# B&R Automation Studio project CControl (part 2)

### Global.var
```iecst
VAR
	Boxen : {REDUND_UNREPLICABLE} fbBoxenKonfig; (*Baustein Trocknungsboxen*)
	Aktoren : {REDUND_UNREPLICABLE} typAktoren; (*Funktionsbausteine aller Aktoren (Ventilatoren, Trocknungsgeräte, Klappen, ...)*)
	Tarifabschaltung : {REDUND_UNREPLICABLE} fbTrockTarifabsch; (*Funktionsbaustein Tarifabschaltung*)
	Strombegrenzung : {REDUND_UNREPLICABLE} fbTrockStrombegr; (*Funktionsbaustein Strombegrenzung*)
END_VAR
VAR RETAIN
	Betriebsparameter : {REDUND_UNREPLICABLE} parAnlage; (*Betriebsparametersatz*)
END_VAR
VAR
	CONST_ZEIT_TESTPHASE : {REDUND_UNREPLICABLE} USINT := 3; (*max. Betriebsstunden, in denen der Kompressor am Luftentfeuchter gestartet werden kann, ohne dass die Mindestlaufzeit der Ölsumpfheizung abgelaufen ist (Für Inbetriebnahme Kältetechniker)*)
	gModul2Vorhanden : {REDUND_UNREPLICABLE} BOOL; (*Variable wird gesetzt, wenn eine Luftentfeuchter-Type mit 2 Kompressormodulen ausgewählt wird*)
	gAktModus : {REDUND_UNREPLICABLE} enumBetriebsmodus; (*Aktueller Schrittkettenzustand*)
	gStatusAnlage : {REDUND_UNREPLICABLE} statAnlage; (*Anlagenstatus*)
	gCmdAnlage : {REDUND_UNREPLICABLE} cmdAnlage; (*Anlagenkommandos*)
END_VAR
VAR RETAIN
	Nutzungsdaten : {REDUND_UNREPLICABLE} typNutzungsdaten; (*Struktur Betriebsstunden, Brennstoffleistung, etc...*)
END_VAR
VAR
	Echtzeit : {REDUND_UNREPLICABLE} typEchtzeit; (*Echtzeituhr*)
	Systeminfo : {REDUND_UNREPLICABLE} typSysteminfo; (*Struktur Systeminformationen (Batteriestatus, Hardwaremodule, etc...)*)
	DateTime : {REDUND_UNREPLICABLE} DATE_AND_TIME; (*Aktuelle Systemzeit*)
	VERSION : {REDUND_UNREPLICABLE} STRING[16] := 'V2.1.3'; (*Softwareversion*)
END_VAR
VAR RETAIN
	gMindestlaufzOelsumpfOk : {REDUND_UNREPLICABLE} BOOL; (*Variable wird gesetzt, wenn Mindestlaufzeit der Ölsumpfheiung abgelaufen ist.*)
END_VAR
VAR
	gAktuellesPasswort : {REDUND_UNREPLICABLE} UDINT; (*Aktuelles Passwort in der Visu (Benutzeranmeldung)*)
	gWerksparameterLaden : {REDUND_UNREPLICABLE} BOOL; (*Befehl Werksparametersatz laden*)
	gEnergiemessungModulOk : {REDUND_UNREPLICABLE} BOOL; (*Modulüberwachung Energiemessmodul (wird in den IO-Mappings zur Fehlergenerierung verwendet)*)
END_VAR
```

### versionsinfo.txt
```
##########################################################
LaTronic CControl 3.07, 4.07 & 4.07 Plus Versionshistorie
##########################################################

--------------------------------------------------------------------------------------------
Version 0.0.0	     	Initialversion			2022.05.19					RL
--------------------------------------------------------------------------------------------

--------------------------------------------------------------------------------------------
Version 0.0.1	     	new/change/fix			2022.06.01					RL
--------------------------------------------------------------------------------------------

Neu:
****
- Optionen für Verhalten der Ventilatoren bei Klappenumschaltungen hinzugefügt (Beide oder nur zuständigen Ventilator
bei Umschaltungen Boxenklappen, Umluftklappen und Bypassklappe).
- Option "Abluftklappe im Frischluftbetrieb immer offen" hinzugefügt (Abluftklappe öffnet im Frischluftbetrieb unabhängig von der
eingestellten Abluftfeuchte, wenn Klappe auf Automatik gestellt).
- Option "Alle Boxenklappen im Stillstand schließen" hinzugefügt.
- Trockengut "Mais" und "Getreide" hinzugefügt.
- VNC-Viewer bei allen Konfigurationen hinzugefügt.
- "Notbetrieb" für alle Boxen und Ventilatoren hinzugefügt (für Auskühlphase Warmluftofen). Boxenklappen und Ventilatoren bleiben aktiv,
bis Auskühlphase abgeschlossen ist.
- Funktion zum Kopieren der XML-Parametersätze auf einen USB-Stick hinzugefügt.
- Zusatztexte hinzugefügt, wenn Trocknungsgeräte wegen Tarifabschaltung aus sind (Vorlaufzeit Tarifabschaltung).
- Zoom für Trendkurven hinzugefügt.
- Hopfen und Kräuter bei Trockengütern hinzugefügt.
- Automatisches Laden der Werksparameter bei neuen Displays hinzugefügt.
- Französische Sprache hinzugefügt.
- Energiemessmodul in allen Hardwarekonfigurationen hinzugefügt.
- Trockengut "Holz" hinzugefügt (Visualisierung/Visu, hmiMain).
- Modulüberwachungen für alle Hardwarekonfigurationen hinzugefügt (IO/io307, io407, io407Plus).

Änderungen:
***********
- Wenn Strombegrenzung der Ventilatoren aktiv ist (Zeitfenster oder digitaler Eingang), geht der Luftentfeuchter bei Überschreiten
des max. Hochdrucks in den Standby-Betrieb (wie bei Klappenumschaltungen).
- Warnung "Entfeuchter Hochdruck max." wird nur generiert, wenn keine Strombegrenzung oder Klappenumschaltung aktiv ist.
- Nur Option "Abluftklappe" ODER "Abluftventilator" erlauben, beide Optionen sind nicht möglich.
- Beim Abschalten der Ventilatoren die Freigabe erst wegschalten, wenn Min-Drehzahl erreicht wurde.
- Buttons und Slider für Ausstattung und Konfiguration Aktoren Boxen sperren, wenn Benutzerebene < LASCO.
- Beim Wechsel von Betrieb auf AUS einer Box -> Arrays Zeitfenster Intervallbetrieb und Nachtrockung auf 0 setzen.
- Entfeuchter, Warmluftofen und Heizregister erst freigeben, wenn zuständiger Ventilator in Betrieb ist.
- Boxen können auch gestartet werden, wenn Summenfehler aktiv (Sperren Visu entfernt, Wechsel in Betriebsart "BETRIEB" trotz Summenfehler).
- Signal "cmdAnlage.FehlerStopp" entfernt (Trocknung kann trotz Fehler gestartet werden bzw. wird nicht mehr automatisch gestoppt).
- Ansteuerung Bypassklappe geändert (actionBetrieb).
- Skalierung Drehzahlvorgabe Kompressor Modul 1 und 2: Min auf "0" gesetzt. (IO/io307, io407Plus).
- Drehzahlvorgaben von FU Kompressor angepasst (Libaries/LascoEntfV2/fbEntfKompressor).
- Doppelmodul nur bei bei den Typen 7, 8, 9 und 10 (10 ist Reserve) (IO/aktorenMapping).
- Fehlermeldungen Entfeuchter Temperatur Eintritt Min/Max nur ausgeben, wenn Entfeuchter angefordert. (Alarmsystem/Alarm).
- Drehzahlvorgabe Heizregister auf Min. setzen, wenn Heizregister nicht freigegeben (Regelung/Leistung).
- Ventilatoren: Wenn eingestellte Drehzahl bei Klappenumschaltungen auf MIN (30%) -> Ventilator ausschalten (Libaries/LascoBoxen/fbBoxenVentKlappen).
- Automatikbetrieb von Abluftklappe auch im Stillstand aktivieren (Ablaufsteuerung/actionStillstand).
- Parameter "Hochdruck Max." und "Verzögerung Standy, wenn Hochdruck Max." bereits ab Benutzerebene "LASCO" einstellbar (Visualisierung/Visu).

Fehlerbehebungen:
*****************
- Indexe für Fehler, Systemmeldungen und Warnungen angepasst (für Filter bei historischen Alarmen).
- Fehler Laufzeitüberwachungen Boxenklappen nur generieren, wenn Klappe verwendet wird.
- Min/Max Werte bei Eingabefeldern Detailansicht Klappen hinzugefügt.
- Struktur "hmiAktuell" remanent deklariert, da ansonsten die Betriebsart der Box nach Stromausfall geändert wird.
- Taste "Datenaufzeichnung auf USB kopieren" zurücksetzen, wenn Kopiervorgang fertig.
- Diverse CSV-Variablen in Datencontainer aktualisiert.
- 4.07Plus: Signalart Luftgeschwindigkeitssensor auf 0-10V geändert.
- Restlaufzeit Ölsumpfheizung in hmiParameter speichern (war Betriebsparameter).
- 4.07 Plus: DO Freigabe Ventilator 2 von Ausgang 2 auf 1 geändert.
- Doppelbelegung von Funktionsbausteinen entfernt (Alarmsystem/Alarm).
- Zusatztext "Auskühlzeit Scheitholzofen" Fehlerbehebung (Visualisierung/hmiConnect).
- Zusatztext "Warten bis Entfeuchter im Stillstand" auch anzeigen, wenn Boxen pausiert werden (Visualisierung/hmiConnect).
- Status Umluftklappen "Aktiv" nur generieren, wenn Klappe in Ausstattung vorhanden (IO/aktorenMapping).
- Digitale Eingänge "diOeldruckKompressorModul2" und "diKopftemperaturKompressorModul2" ausgetauscht (IO/io407Plus).
- Eingang "BetriebsmeldungVent" von Kompressor Modul 2 korrigiert (IO/aktorenMapping).
- "StoerungOut" von Funktionsbaustein "fbEntfKompressor" nicht automatisch rücksetzen, muss manuell quittiert werden (Libaries/LaEntfV2/fbEntfKompressor).
- Digialen Eingang "BetriebsmldgKompressorMod1" im IO-Test korrigiert (IO/io407Plus).
- 3.07: Je nach Ausstattung Analogeingänge und Statuseingänge als Dachluft- oder Frischluftsensor skalieren (IO/io307).

--------------------------------------------------------------------------------------------
Version 1.0.0	     	Erstversion Auslieferung		2022.06.22					RL
--------------------------------------------------------------------------------------------

--------------------------------------------------------------------------------------------
Version 1.1.0	     	new/fix/change					2022.09.22					RL
--------------------------------------------------------------------------------------------

Neu:
****
- Slowenische Sprache hinzugefügt (Visualisierung).
- Laden und Erstellen eines Parametersatzes sperren, wenn Filename "307Werk", "407Werk" oder "407PlusWerk" ist (Visualisierung/Visu).

Änderungen:
***********
- Die letzten 100 Ereignisse in der Alarmhistorie werden remanent aufgezeichnet (Visualisierung/Visu).

Fehlerbehebungen:
*****************
- Temperatur Austritt Entfeuchter: Falsch angehängten Wert in Visu korrigiert (Visualisierung/hmiMain).

TODO:
*****
- Verzögerungszeit Umschaltung Klappen, bis Endlage erreicht wurde?

--------------------------------------------------------------------------------------------
Version 1.1.1	     	fix								2022.09.22					RL
--------------------------------------------------------------------------------------------

Fehlerbehebungen:
*****************
- Bei Anlagen mit Bypassklappe: Freigabe Entfeuchter war von Betrieb des zuständigen Ventilators abhängig. Dadurch war die Freigabe des Kompressors immer nur solange
vorhanden, bis die Bypassklappe umgeschaltet wurde (ständiges hin- und herschalten der Klappen). Geändert, dass die Kompressor-Freigabe erhalten bleibt, wenn die Ventilatoren
kurzzeitig zum Umschalten der Klappen ausgeschaltet werden (Ablaufsteuerung/Ablaufstrg/actionBetrieb).

--------------------------------------------------------------------------------------------
Version 1.1.2	     	new								2023.05.03					RL
--------------------------------------------------------------------------------------------

Neu:
****
- Sensor Kanaldruck für Konfiguration 3.07 hinzugefügt (IO/io307).

--------------------------------------------------------------------------------------------
Version 1.2.0	     	new/change						2023.05.26					RL
--------------------------------------------------------------------------------------------

Neu:
****
- Neue Visualisierung für CControl 3.04 hinzugefügt (PPC30 4 Zoll).
- Hardwarekonfiguration & IO-mapping für CControl 3.04 hinzugefügt.
- Ausgänge öffnen/schliessen für Klappenansteuerungen (Umluftklappen, Bypassklappe, Abluftklappe, ...) hinzugefügt.
- Inselbetrieb für Luftentfeuchter hinzugefügt.

Änderungen:
***********
- Statuseingang "rel. Feuchte MAX" bei allen Feuchte/Temperaturfühlern für Fehlergenerierung entfernt (führt ansonsten zu Fehler, wenn rel. Feuchte tatsächlich bei 100% ist) (Alarmsystem/Alarm)

--------------------------------------------------------------------------------------------
Version 2.0.0	     	new/change						2024.07.04					RL
--------------------------------------------------------------------------------------------

Neu:
****
- Konfiguration für HB4000 & HB3000 hinzugefügt.
- Betriebsmodus "Dauerbetrieb" in "Automatik" umbenannt. Bei Anlagen ohne Luftaufbereitung (Kaltbelüftungen) wechselt die Box
bei schlechter Witterung in einen Puls/Pausebetrieb (wie bei HB3000/HB4000). Die Bestimmung der Witterungsverhältnisse kann für jede
Box seperat eingestellt werden.
- Entfeuchter Fremdgerät hinzugefügt (Ansteuerung von Frigopol/Baier Luftentfeuchtern).
- Option für Stellung Umluftklappen im Stillstand (Frischluft oder Umluft), wenn Umluftklappen im Automatikbetrieb sind.
- Option "Endlagen" für alle Klappenantriebe (ausgenommen Abluftklappe) hinzugefügt. Wird die Option ausgeschaltet (keine Endlagen vorhanden), wird über die
eingestellte Laufzeit der Klappe die Fahrt simuliert (Ventilator bleibt für die Laufzeit ausgeschaltet/reduziert).

Änderungen:
***********
- Im Stillstand Umluftklappen & Abluftklappe nicht automatisch umschalten (Ablaufsteuerung, Ablaufstrg/actionBetrieb).
- Default-Gateway als DEV1-Port verwenden (war fix auf 10.0.0.1 eingestellt) (Sitemanager/Sitemanager).
- Parameter "Einschaltverzögerung Entfeuchter" von 30 auf 120 Sekunden im Standardparametersatz aller Entfeuchtersteuerungen geändert (lt. Werner).

TODO:
*****
- Übersetzungen ergänzen (Aktuell nur Deutsch und Englisch verfügbar)
- Visu 3.04
- Standardparameter restliche Steuerungen

--------------------------------------------------------------------------------------------
Version 2.1.0	     	new/change						2024.12.02					RL
--------------------------------------------------------------------------------------------

Neu:
****
- Option Stellung Umluftklappen im Stillstand: Stellung kann für Klappe 1 und 2 separat eingestellt werden.
- Konfiguration für CControl 2.07 hinzugefügt.

Änderungen:
***********
- Schlechtwetterbetrieb: Anstatt der Boxenlaufzeit (in Stunden) wird die aktuelle Stufe durch die Trockengutfeuchte (%) bestimmt (manuelle Eingabe durch Bediener).

--------------------------------------------------------------------------------------------
Version 2.1.1	     	new/change						2025.05.07					RIG
--------------------------------------------------------------------------------------------

Änderungen:
***********
- Bugfix - Bei der Karte X20CM8281f war die Modulueberwachung aktiviert. Dies fuehrte dazu das die Steuerung nicht hochgefahren ist und beim Booten im Servicemodus haengen blieb.

--------------------------------------------------------------------------------------------
Version 2.1.2	     	new/change						2025.05.15					RIG
--------------------------------------------------------------------------------------------

Änderungen:
***********
- Bugfix - Fehler Betriebsmeldung "Entfeuchter Fremdgerät" wurde gesetzt obwohl Fremdgeraet nicht aktiviert war

--------------------------------------------------------------------------------------------
Version 2.1.3	     	new/change						2025.06.12					RIG
--------------------------------------------------------------------------------------------

Neu:
****
- Parametersaetze fuer 3.04 und 3.07 erstellt. Wurden aus 4.07 kopiert!
- Registerflache <Property ID="[2]" DataType="REAL" Value="3.3" /> von 3.8 auf 3.3 geaendert. Laut Werner war das schon immer falsch.

Änderungen:
***********
- Bugfix - Klappenansteuerung Anzugsverzoegerung fuer oeffnen und schliessen der Klappen eingebaut. Dient dazu das andere Relaise abfallen zu lassen bevor das andere geschaltet wird. Verhindert Doppelansteuerung.
```

### Program Logical/Alarmsystem/Alarm

#### AlarmCyclic.st
```iecst
PROGRAM _INIT

	init	:= FALSE;

END_PROGRAM

PROGRAM _CYCLIC

	//Sekundentick generieren
	//=======================
	eUhr(Freigabe:= TRUE);
	fbLascoZdxx_0(IN := eUhr.Sekunde);
	sekTick	:= fbLascoZdxx_0.Q;

	//Fehlergenerierung eingeschaltet *****************************************************************************************************************************************************************
	IF init THEN

		//=======================================================================================================================================================
		//FEHLER ------------------------------ FEHLER ------------------------------ FEHLER ------------------------------ FEHLER ------------------------------
		//=======================================================================================================================================================

		//00) Fehler Absicherung 24VDC
		alarmFehler[FEHLER_24VDC]			:= NOT di24VDCinternIstOk;

		//01) Fehler FU Kompressor Modul 1
		alarmFehler[FEHLER_FU_KOMPRESSOR_MODUL1]	:= Aktoren.KompressorModul1.StoerungOut;

		//02) Fehler FU Kompressor Modul 2
		alarmFehler[FEHLER_FU_KOMPRESSOR_MODUL2]	:= Aktoren.KompressorModul2.StoerungOut;

		//03) Fehler Betriebsmeldung Kompressor Modul 1
		fbLascoFehl_0(FehlerIn := doKompressorEinModul1 AND NOT diBetriebsmldgKompressorModul1,
		VerzZeit := Betriebsparameter.Allgemein.VerzoegerungFehler, Quit := hmiButtons.QuitFehler, Tick := sekTick, Mode := 1);
		alarmFehler[FEHLER_BETRIEBSMLDG_KOMPR_MOD1]	:= fbLascoFehl_0.FehlerOut;

		//04) Fehler Betriebsmeldung Kompressor Modul 2
		fbLascoFehl_1(FehlerIn := gModul2Vorhanden AND doKompressorEinModul2 AND NOT diBetriebsmldgKompressorModul2,
		VerzZeit := Betriebsparameter.Allgemein.VerzoegerungFehler, Quit := hmiButtons.QuitFehler, Tick := sekTick, Mode := 1);
		alarmFehler[FEHLER_BETRIEBSMLDG_KOMPR_MOD2]	:= fbLascoFehl_1.FehlerOut;

		//05) Fehler Betriebsmeldung Ventilator 1
		fbLascoFehl_2(FehlerIn := Aktoren.VentUndKlappen.FehlerFuVentilator1,
		VerzZeit := 0, Quit := hmiButtons.QuitFehler, Tick := sekTick, Mode := 1);
		alarmFehler[FEHLER_BETRIEBSMLDG_VENTILATOR1]	:= fbLascoFehl_2.FehlerOut;

		//06) Fehler Betriebsmeldung Ventilator 2
		fbLascoFehl_3(FehlerIn := Aktoren.VentUndKlappen.FehlerFuVentilator2,
		VerzZeit := 0, Quit := hmiButtons.QuitFehler, Tick := sekTick, Mode := 1);
		alarmFehler[FEHLER_BETRIEBSMLDG_VENTILATOR2]	:= fbLascoFehl_3.FehlerOut;

		//07) Fehler Betriebsmeldung Abluftventilator
		fbLascoFehl_4(FehlerIn := Aktoren.Abluftventilator.FehlerOut,
		VerzZeit := 0, Quit := hmiButtons.QuitFehler, Tick := sekTick, Mode := 1);
		alarmFehler[FEHLER_BETRIEBSMLDG_ABLUFTVENT]	:= fbLascoFehl_4.FehlerOut;

		//08) Fehler Hochdruck Modul 1
		fbLascoFehl_5(FehlerIn :=  Betriebsparameter.Ausstattung.Entfeuchter AND NOT diHochdruckOkModul1, VerzZeit := 0,
		Quit := hmiButtons.QuitFehler, Tick := sekTick, Mode := 0);
		alarmFehler[FEHLER_HOCHDRUCK_MODUL1]			:= fbLascoFehl_5.FehlerOut;

		//09) Fehler Hochdruck Modul 2
		fbLascoFehl_6(FehlerIn :=  Betriebsparameter.Ausstattung.Entfeuchter AND gModul2Vorhanden AND NOT diHochdruckOkModul2, VerzZeit := 0,
		Quit := hmiButtons.QuitFehler, Tick := sekTick, Mode := 0);
		alarmFehler[FEHLER_HOCHDRUCK_MODUL2]			:= fbLascoFehl_6.FehlerOut;

		//10) Fehler Niederdruck Modul 1
		fbLascoFehl_7(FehlerIn := Betriebsparameter.Ausstattung.Entfeuchter AND NOT diNiederdruckOkModul1, VerzZeit := 0,
		Quit := hmiButtons.QuitFehler, Tick := sekTick, Mode := 0);
		alarmFehler[FEHLER_NIEDERDRUCK_MODUL1]			:= fbLascoFehl_7.FehlerOut;

		//11) Fehler Niederdruck Modul 2
		fbLascoFehl_8(FehlerIn := Betriebsparameter.Ausstattung.Entfeuchter AND gModul2Vorhanden AND NOT diNiederdruckOkModul2,
		VerzZeit := 0, Quit := hmiButtons.QuitFehler, Tick := sekTick, Mode := 0);
		alarmFehler[FEHLER_NIEDERDRUCK_MODUL2]			:= fbLascoFehl_8.FehlerOut;

		//12) Fehler Öldruck Kompressor Modul 1
		fbLascoFehl_9(FehlerIn := Betriebsparameter.Ausstattung.Entfeuchter AND NOT diOeldruckKompressorModul1,
		VerzZeit := 0, Quit := hmiButtons.QuitFehler, Tick := sekTick, Mode := 0);
		alarmFehler[FEHLER_OELDRUCK_KOMPR_MOD1]			:= fbLascoFehl_9.FehlerOut;

		//13) Fehler Öldruck Kompressor Modul 2
		fbLascoFehl_10(FehlerIn := Betriebsparameter.Ausstattung.Entfeuchter AND gModul2Vorhanden AND NOT diOeldruckKompressorModul2,
		VerzZeit := 0, Quit := hmiButtons.QuitFehler, Tick := sekTick, Mode := 0);
		alarmFehler[FEHLER_OELDRUCK_KOMPR_MOD2]			:= fbLascoFehl_10.FehlerOut;

		//14) Fehler Kopftemperatur Kompressor Modul 1
		fbLascoFehl_11(FehlerIn := Betriebsparameter.Ausstattung.Entfeuchter AND NOT diKopftempKompressorModul1,
		VerzZeit := 0, Quit := hmiButtons.QuitFehler, Tick := sekTick, Mode := 0);
		alarmFehler[FEHLER_KOPFTEMP_KOMPR_MOD1]			:= fbLascoFehl_11.FehlerOut;

		//15) Fehler Kopftemperatur Kompressor Modul 2
		fbLascoFehl_12(FehlerIn := Betriebsparameter.Ausstattung.Entfeuchter AND gModul2Vorhanden AND NOT diKopftempKompressorModul2,
		VerzZeit := 0, Quit := hmiButtons.QuitFehler, Tick := sekTick, Mode := 0);
		alarmFehler[FEHLER_KOPFTEMP_KOMPR_MOD2]			:= fbLascoFehl_12.FehlerOut;

		//16) Fehler Vollschutz Kompressor Modul 1
		fbLascoFehl_13(FehlerIn := Betriebsparameter.Ausstattung.Entfeuchter AND NOT diVollschutzKompressorModul1,
		VerzZeit := 0, Quit := hmiButtons.QuitFehler, Tick := sekTick, Mode := 0);
		alarmFehler[FEHLER_VOLLSCHUTZ_KOMPR_MOD1]			:= fbLascoFehl_13.FehlerOut;

		//17) Fehler Vollschutz Kompressor Modul 2
		fbLascoFehl_14(FehlerIn := Betriebsparameter.Ausstattung.Entfeuchter AND gModul2Vorhanden AND NOT diVollschutzKompressorModul2,
		VerzZeit := 0, Quit := hmiButtons.QuitFehler, Tick := sekTick, Mode := 0);
		alarmFehler[FEHLER_VOLLSCHUTZ_KOMPR_MOD2]			:= fbLascoFehl_14.FehlerOut;

		//18) Fehler Betriebsmeldung Warmluftofen
		alarmFehler[FEHLER_BETRIEBSMLDG_WARMLUFTOFEN]	:= Aktoren.Warmluftofen.FehlerBetriebsmeldungOut;

		//19) Fehler Betriebsmeldung Notstromaggregat
		alarmFehler[FEHLER_BETRIEBSMLDG_NOTSTROM]		:= Aktoren.Notstromaggregat.FehlerOut;

		//20 - 31) Sensoren
		fbLascoFehl_15(FehlerIn := ((*diStatusFrischluftFeuchteMax OR *)diStatusFrischluftFeuchteMin OR diStatusFrischluftTempMax OR diStatusFrischluftTempMin) AND
		Betriebsparameter.Ausstattung.SensorFrischluft, VerzZeit := Betriebsparameter.Allgemein.VerzoegerungFehler,
		Quit := hmiButtons.QuitFehler, Tick := sekTick, Mode := 1);
		alarmFehler[FEHLER_SENSOR_FRISCHLUFT]	:= fbLascoFehl_15.FehlerOut;

		fbLascoFehl_16(FehlerIn := ((*diStatusDachluftFeuchteMax OR *)diStatusDachluftFeuchteMin OR diStatusDachluftTempMax OR diStatusDachluftTempMin) AND
		Betriebsparameter.Ausstattung.SensorDachluft, VerzZeit := Betriebsparameter.Allgemein.VerzoegerungFehler,
		Quit := hmiButtons.QuitFehler, Tick := sekTick, Mode := 1);
		alarmFehler[FEHLER_SENSOR_DACHLUFT]	:= fbLascoFehl_16.FehlerOut;

		fbLascoFehl_17(FehlerIn := ((*diStatusTrockenluftFeuchteMax OR *)diStatusTrockenluftFeuchteMin OR diStatusTrockenluftTempMax OR diStatusTrockenluftTempMin) AND
		Betriebsparameter.Ausstattung.SensorTrockenluft, VerzZeit := Betriebsparameter.Allgemein.VerzoegerungFehler,
		Quit := hmiButtons.QuitFehler, Tick := sekTick, Mode := 1);
		alarmFehler[FEHLER_SENSOR_TROCKENLUFT]	:= fbLascoFehl_17.FehlerOut;

		fbLascoFehl_18(FehlerIn := ((*diStatusAbluftFeuchteMax OR *)diStatusAbluftFeuchteMin OR diStatusAbluftTempMax OR diStatusAbluftTempMin) AND
		Betriebsparameter.Ausstattung.SensorAbluft,VerzZeit := Betriebsparameter.Allgemein.VerzoegerungFehler,
		Quit := hmiButtons.QuitFehler, Tick := sekTick, Mode := 1);
		alarmFehler[FEHLER_SENSOR_ABLUFT]	:= fbLascoFehl_18.FehlerOut;

		fbLascoFehl_19(FehlerIn := Betriebsparameter.Ausstattung.Entfeuchter AND
		((*diStatusEintrittFeuchteMax OR *)diStatusEintrittFeuchteMin OR diStatusEintrittTempMax OR diStatusEintrittTempMin),
		VerzZeit := Betriebsparameter.Allgemein.VerzoegerungFehler, Quit := hmiButtons.QuitFehler, Tick := sekTick, Mode := 1);
		alarmFehler[FEHLER_SENSOR_EINTRITT]	:= fbLascoFehl_19.FehlerOut;

		alarmFehler[FEHLER_SENSOR_AUSTRITT]	:= FALSE;	//Fehler Sensor Austritt nur als Warnung generieren

		fbLascoFehl_20(FehlerIn := (diStatusLuftgeschwDrahtbruch OR diStatusLuftgeschwMax OR diStatusLuftgeschwMin) AND Betriebsparameter.Ausstattung.SensorLuftgeschwindigkeit,
		VerzZeit := Betriebsparameter.Allgemein.VerzoegerungFehler, Quit := hmiButtons.QuitFehler, Tick := sekTick, Mode := 1);
		alarmFehler[FEHLER_SENSOR_LUFTGESCHW]	:= fbLascoFehl_20.FehlerOut;

		fbLascoFehl_21(FehlerIn := (diStatusDifferenzdruckMax OR diStatusDifferenzdruckMin) AND Betriebsparameter.Ausstattung.SensorKanaldruck,
		VerzZeit := Betriebsparameter.Allgemein.VerzoegerungFehler, Quit := hmiButtons.QuitFehler, Tick := sekTick, Mode := 1);
		alarmFehler[FEHLER_SENSOR_KANALDRUCK]	:= fbLascoFehl_21.FehlerOut;

		fbLascoFehl_22(FehlerIn := Betriebsparameter.Ausstattung.Entfeuchter AND (diStatusNiederdruckMaxMod1 OR diStatusNiederdruckMinMod1),
		VerzZeit := Betriebsparameter.Allgemein.VerzoegerungFehler, Quit := hmiButtons.QuitFehler, Tick := sekTick, Mode := 1);
		alarmFehler[FEHLER_SENSOR_NIEDERDRUCK_MOD1]	:= fbLascoFehl_22.FehlerOut;

		fbLascoFehl_23(FehlerIn := Betriebsparameter.Ausstattung.Entfeuchter AND gModul2Vorhanden AND (diStatusNiederdruckMaxMod2 OR diStatusNiederdruckMinMod2),
		VerzZeit := Betriebsparameter.Allgemein.VerzoegerungFehler, Quit := hmiButtons.QuitFehler, Tick := sekTick, Mode := 1);
		alarmFehler[FEHLER_SENSOR_NIEDERDRUCK_MOD2]	:= fbLascoFehl_23.FehlerOut;

		fbLascoFehl_24(FehlerIn := Betriebsparameter.Ausstattung.Entfeuchter AND (diStatusHochdruckMaxMod1 OR diStatusHochdruckMinMod1),
		VerzZeit := Betriebsparameter.Allgemein.VerzoegerungFehler, Quit := hmiButtons.QuitFehler, Tick := sekTick, Mode := 1);
		alarmFehler[FEHLER_SENSOR_HOCHDRUCK_MOD1]	:= fbLascoFehl_24.FehlerOut;

		fbLascoFehl_25(FehlerIn := Betriebsparameter.Ausstattung.Entfeuchter AND gModul2Vorhanden AND (diStatusHochdruckMaxMod2 OR diStatusHochdruckMinMod2),
		VerzZeit := Betriebsparameter.Allgemein.VerzoegerungFehler, Quit := hmiButtons.QuitFehler, Tick := sekTick, Mode := 1);
		alarmFehler[FEHLER_SENSOR_HOCHDRUCK_MOD2]	:= fbLascoFehl_25.FehlerOut;

		//32) Fehler Endlagen Bypassklappe
		alarmFehler[FEHLER_ENDLAGEN_BYPASSKLAPPE]		:= Aktoren.VentUndKlappen.FehlerLaufzeitBypass AND Betriebsparameter.Ausstattung.Bypassklappe;

		//33) Fehler Endlagen Umschaltklappe 1
		alarmFehler[FEHLER_ENDLAGEN_UMSCHALTKLAPPE1]	:= Aktoren.VentUndKlappen.FehlerLaufzeitUmschaltkl1 AND Betriebsparameter.Ausstattung.Umschaltklappe1;

		//34) Fehler Endlagen Umschaltklappe 2
		alarmFehler[FEHLER_ENDLAGEN_UMSCHALTKLAPPE2]	:= Aktoren.VentUndKlappen.FehlerLaufzeitUmschaltkl2 AND Betriebsparameter.Ausstattung.Umschaltklappe2;

		//35) Fehler Endlagen Boxenklappe 1
		alarmFehler[FEHLER_ENDLAGEN_BOXENKLAPPE_1]		:= Aktoren.VentUndKlappen.FehlerLaufzeitKlappeBox1;

		//36) Fehler Endlagen Boxenklappe 2
		alarmFehler[FEHLER_ENDLAGEN_BOXENKLAPPE_2]		:= Aktoren.VentUndKlappen.FehlerLaufzeitKlappeBox2;

		//37) Fehler Endlagen Boxenklappe 3
		alarmFehler[FEHLER_ENDLAGEN_BOXENKLAPPE_3]		:= Aktoren.VentUndKlappen.FehlerLaufzeitKlappeBox3;

		//38) Fehler Endlagen Boxenklappe 4
		alarmFehler[FEHLER_ENDLAGEN_BOXENKLAPPE_4]		:= Aktoren.VentUndKlappen.FehlerLaufzeitKlappeBox4;

		//39) Fehler Endlagen Boxenklappe 5
		alarmFehler[FEHLER_ENDLAGEN_BOXENKLAPPE_5]		:= Aktoren.VentUndKlappen.FehlerLaufzeitKlappeBox5;

		//40) Fehler Endlagen Boxenklappe 6
		alarmFehler[FEHLER_ENDLAGEN_BOXENKLAPPE_6]		:= Aktoren.VentUndKlappen.FehlerLaufzeitKlappeBox6;

		//41) Fehler Endlagen Abluftklappe
		alarmFehler[FEHLER_ENDLAGEN_ABLUFTKLAPPE]		:= Aktoren.Abluftklappe.FehlerLaufzeit;

		//42) Fehler Temperatur Eintritt zu hoch
		alarmFehler[FEHLER_EINTRITT_TEMP_ZU_HOCH]		:= (gStatusAnlage.EintrittTemperatur > Betriebsparameter.Kompressor1.EintrittTempMax) AND
		Betriebsparameter.Ausstattung.Entfeuchter AND Boxen.FreigabeLuftentfeuchter;

		//43) Fehler Temperatur Eintritt zu niedrig
		alarmFehler[FEHLER_EINTRITT_TEMP_ZU_NIEDRIG]	:= (gStatusAnlage.EintrittTemperatur < Betriebsparameter.Kompressor1.EintrittTempMin) AND
		Betriebsparameter.Ausstattung.Entfeuchter AND Boxen.FreigabeLuftentfeuchter;

		//44) Fehler Laufzeit Pumpdown Kompressor Modul 1
		alarmFehler[FEHLER_LZ_PUMPDOWN_MOD1]			:= Aktoren.KompressorModul1.FehlerPumpdown;

		//45) Fehler Laufzeit Pumpdown Kompressor Modul 2
		alarmFehler[FEHLER_LZ_PUMPDOWN_MOD2]			:= Aktoren.KompressorModul2.FehlerPumpdown AND gModul2Vorhanden;

		//46) Drehfeldüberwachung (Nur bei 3.04 Plus vorhanden)
		IF hmiStatus.NameSteuerung = 3 THEN
			alarmFehler[FEHLER_DREHFELD]	:= NOT diDrehfeldIstKorrekt AND NOT alarmSystem[FEHLER_KOMMUNIKATION_DISPLAY_IO];
		ELSE
			alarmFehler[FEHLER_DREHFELD]	:= FALSE;
		END_IF

		//47) Störmeldung Entfeuchter Fremdgeräte
		fbLascoFehl_29(FehlerIn := Betriebsparameter.Ausstattung.EntfeuchterFremd AND diEntfeuchterFremdStoerung,
		VerzZeit := Betriebsparameter.Allgemein.VerzoegerungFehler, Quit := hmiButtons.QuitFehler, Tick := sekTick, Mode := 2);
		alarmFehler[FEHLER_ENTF_FREMD_STOERMELDUNG]			:= fbLascoFehl_29.FehlerOut;

		//48) Fehler Betriebsmeldung Entfeuchter Fremdgerät
		alarmFehler[FEHLER_ENTF_FREMD_BETRMLDG]			:= Betriebsparameter.Ausstattung.EntfeuchterFremd AND Aktoren.EntfeuchterFremd.FehlerBetriebsmldg; //V2.1.2

		//=======================================================================================================================================================
		//WARNUNGEN ------------------------------ WARNUNGEN ------------------------------ WARNUNGEN ------------------------------ WARNUNGEN ------------------
		//=======================================================================================================================================================

		//00) Warnung wenn Hochdruck Modul 1 zu hoch (Register verschmutzt, Ansaugtemperatur zu hoch oder zu wenig Luftmenge
		fbLascoFehl_26(FehlerIn := gStatusAnlage.Betrieb AND (gStatusAnlage.HochdruckModul1 > Betriebsparameter.Kompressor1.HochdruckMax) AND NOT
		Aktoren.KompressorModul1.KlappenumschaltungAkiv,
		VerzZeit := Betriebsparameter.Allgemein.VerzoegerungWarnungen, Quit := hmiButtons.QuitFehler, Tick := sekTick, Mode := 0);
		alarmWarnung[WARNUNG_HOCHDRUCK_MAX_MOD1]	:= fbLascoFehl_26.FehlerOut;

		//01) Warnung wenn Hochdruck Modul 2 zu hoch (Register verschmutzt, Ansaugtemperatur zu hoch oder zu wenig Luftmenge
		fbLascoFehl_27(FehlerIn := gModul2Vorhanden AND gStatusAnlage.Betrieb AND
		(gStatusAnlage.HochdruckModul2 > Betriebsparameter.Kompressor1.HochdruckMax) AND NOT Aktoren.KompressorModul2.KlappenumschaltungAkiv,
		VerzZeit := Betriebsparameter.Allgemein.VerzoegerungWarnungen, Quit := hmiButtons.QuitFehler, Tick := sekTick, Mode := 0);
		alarmWarnung[WARNUNG_HOCHDRUCK_MAX_MOD2]	:= fbLascoFehl_27.FehlerOut;

		//02) Warnung Sensor Austritt
		fbLascoFehl_28(FehlerIn := diStatusAustrittFeuchteMax OR diStatusAustrittFeuchteMin OR diStatusAustrittTempMax OR diStatusAustrittTempMin,
		VerzZeit := Betriebsparameter.Allgemein.VerzoegerungFehler, Quit := hmiButtons.QuitFehler, Tick := sekTick, Mode := 1);
		alarmWarnung[WARNUNG_SENSOR_AUSTRITT]	:= fbLascoFehl_28.FehlerOut;

		//==================================================================================================================================================================
		//Fehlerausgang
		//==================================================================================================================================================================

		IF (gStatusAnlage.Betrieb OR gAktModus = STILLSTAND) THEN
			doTrocknungStoerung 	:= gStatusAnlage.Fehler.SummeFehler;
		ELSE
			doTrocknungStoerung	:= FALSE;
		END_IF

	END_IF

	//00 - 04 Systemfehler

	//alarmSystem[FEHLER_KOMMUNIKATION_DISPLAY_IO]	:= ; Wird in den IO-Mappings erzeugt.
	alarmSystem[FEHLER_IO_TEST_NICHT_FERTIG]		:= NOT Nutzungsdaten.Allgemein.IoTestAbgeschlossen;

	//Fehlerquittierung rücksetzen
	TON_Fehlerquittierung.IN	:= hmiButtons.QuitFehler;
	TON_Fehlerquittierung.PT	:= UDINT_TO_TIME(CONST_VERZ_QUIT);
	TON_Fehlerquittierung();

	IF (TON_Fehlerquittierung.Q) THEN
		hmiButtons.QuitFehler	:= FALSE;
	END_IF

	//Gruppenalarme bilden
	//********************

	gStatusAnlage.Fehler.SummeFehler := FALSE;
	gStatusAnlage.Fehler.FehlerNr	 := 0;
	ilen := (SIZEOF(alarmFehler) / SIZEOF(alarmFehler[0])) - 1;
	FOR i := 0 TO ilen DO
		IF (alarmFehler[i] = TRUE) THEN
			gStatusAnlage.Fehler.SummeFehler 	:= TRUE;
			gStatusAnlage.Fehler.FehlerNr		:= i + 1;
			EXIT;
		END_IF
	END_FOR

	gStatusAnlage.Fehler.SummeWarnung := FALSE;
	gStatusAnlage.Fehler.WarnungNr		 := 0;
	ilen := (SIZEOF(alarmWarnung) / SIZEOF(alarmWarnung[0])) - 1;
	FOR i := 0 TO ilen DO
		IF (alarmWarnung[i] = 1) THEN
			gStatusAnlage.Fehler.SummeWarnung 	:= TRUE;
			gStatusAnlage.Fehler.WarnungNr		:= i + 1;
			EXIT;
		END_IF
	END_FOR

	gStatusAnlage.Fehler.SummeSystem := FALSE;
	ilen := (SIZEOF(alarmSystem) / SIZEOF(alarmSystem[0])) - 1;
	FOR i := 0 TO ilen DO
		IF (alarmSystem[i] = 1) THEN
			gStatusAnlage.Fehler.SummeSystem := TRUE;
			EXIT;
		END_IF
	END_FOR

	init	:= TRUE;

END_PROGRAM
```

### CSV01_CFG.dat
```
; ============================================================================================
; ACHTUNG: !!! In diesem Datenmodul dürfen absolut keine Tabulator-Sprünge enthalten sein !!!!
; ============================================================================================

;[ABSCHNITT_CONFIG]
;******************

;<----------------->   -> Länge der 8 nachstehenden Eingabefelder
"1.0.0.1            "  ; USINT[0..19] CSV-Version für Auswertung in Reporting-Software                  z.B.: "1.0.0.1            "
"LATronicCControl   "  ; USINT[0..19] Anlagenname                                                       z.B.: "Heizung_01         "
"CF                 "  ; USINT[0..19]          RPS-Ebene: File-Devicename (CPU Eigenschaften)           z.B.: "CF                 "
"CSV                "  ; USINT[0..19]          RPS-Ebene: Zielordner (nur eine Hirachieebene möglich)   z.B.: "CSV                "
"usb_device         "  ; USINT[0..19] [OPTION] EXTERN   : File-Devicename (CPU Eigenschaften)           z.B.: "USB                "
"CSV                "  ; USINT[0..19] [OPTION] EXTERN   : Zielordner (nur eine Hirachieebene möglich)   z.B.: "CSV                "
"192.168.203.202    "  ; USINT[0..19] [OPTION] PC-Ebene : IP-Adresse PC                                 z.B.: "192.168.203.204    "
"PC_D               "  ; USINT[0..19] [OPTION] PC-Ebene : Windows-Freigabename des Laufwerks am PC  	z.B.: "PC_D               "
"guest              "  ; USINT[0..19] [OPTION] PC-Ebene : Windows-Username (nicht akt. Anmeldung verw.) z.B.: "guest              "
"guest              "  ; USINT[0..19] [OPTION] PC-Ebene : Windows-Userpassword                      	z.B.: "guest              "
"/Daten/Excel/CSV                                                                                   " ;USINT[0..99] [OPTION] PC-Ebene: Zielordner (muß am PC manuell angelegt werden
;<------------------------------------------------------------------------------------------------->

;[ABSCHNITT_DATEN]
;*****************

;TAG-ID          TAG-Variablenname (RPS-Name)                                  TAG-Bezeichung                                   TAG-Einheit                  TAG-MIN           TAG-MAX
;[DINT]                USINT[0..47]                                             USINT[0..59]                                    USINT[0..31]                USINT[0..15]      USINT[0..15]
; 0..9999
;(mit "0"          (RPS-Variablenname)                                          (freier Text)                                   (freier Text)               (Komma=".")       (Komma=".")
;auffüllen!)                                                                                                                                               (=Trend SkalaU)    (=Trend SkalaO)
;                                                                                                                                                          (=Def. Kommast.)  (=Def. Kommast.)
;---->  <--------------------------------------------->   <--------------------------------------------------------->   <----------------------------->   <------------->   <------------->
000001,"gStatusAnlage.Betrieb                          ","ALLG: Betrieb Anlage                                       ","0/1                            ","              0","              1"
000002,"gAktuellesPasswort                             ","ALLG: Aktuelles Passwort                                   ","Num                            ","              0","         999999"
000003,"gStatusAnlage.FrischluftbetriebAktiv           ","ALLG: Frischluftbetrieb Aktiv                              ","0/1                            ","              0","              1"
000004,"gStatusAnlage.UmluftbetriebAktiv               ","ALLG: Umluftbetrieb Aktiv                                  ","0/1                            ","              0","              1"
000005,"gStatusAnlage.Fehler.FehlerNr                  ","ALLG: Fehlernummer                                         ","0-39                           ","              0","             39"
000006,"gStatusAnlage.Fehler.WarnungNr                 ","ALLG: Warnungsnummer                                       ","0-29                           ","              0","             29"
000007,"Aktoren.KompressorModul1.curStep               ","ALLG: Aktueller Schritt Kompressor 1                       ","0-6                            ","              0","              6"
000008,"Aktoren.KompressorModul2.curStep               ","ALLG: Aktueller Schritt Kompressor 2                       ","0-6                            ","              0","              6"
000009,"aiNiederdruckModul1                            ","AI: Niederdruck Modul 1                                    ","bar                            ","            0.0","           30.0"
000010,"aiHochdruckModul1                              ","AI: Hochdruck Modul 1                                      ","bar                            ","            0.0","           30.0"
000011,"aiNiederdruckModul2                            ","AI: Niederdruck Modul 2                                    ","bar                            ","            0.0","           30.0"
000012,"aiHochdruckModul2                              ","AI: Hochdruck Modul 2                                      ","bar                            ","            0.0","           30.0"
000013,"aiFrischluftTemperatur                         ","AI: Frischluft Temperatur                                  ","°C                             ","          -30.0","           70.0"
000014,"aiFrischluftFeuchte                            ","AI: Frischluft rel. Feuchte                                ","%                              ","            0.0","          100.0"
000015,"aiDachluftTemperatur                           ","AI: Dachluft Temperatur                                    ","°C                             ","          -30.0","           70.0"
000016,"aiDachluftFeuchte                              ","AI: Dachluft rel. Feuchte                                  ","%                              ","            0.0","          100.0"
000017,"aiTrockenluftTemperatur                        ","AI: Trockenluft Temperatur                                 ","°C                             ","          -30.0","           70.0"
000018,"aiTrockenluftFeuchte                           ","AI: Trockenluft rel. Feuchte                               ","%                              ","            0.0","          100.0"
000019,"aiAbluftTemperatur                             ","AI: Abluft Temperatur                                      ","°C                             ","          -30.0","           70.0"
000020,"aiAbluftFeuchte                                ","AI: Abluft rel. Feuchte                                    ","%                              ","            0.0","          100.0"
000021,"aiLuftgeschwindigkeit                          ","AI: Luftgeschwindikeit                                     ","m/s                            ","            0.0","           20.0"
000022,"aiDifferenzdruck                               ","AI: Kanaldruck                                             ","Pa                             ","            0.0","         5000.0"
000023,"aiEintrittTemperatur                           ","AI: Eintritt Temperatur                                    ","°C                             ","          -30.0","           70.0"
000024,"aiEintrittFeuchte                              ","AI: Eintritt rel. Feuchte                                  ","%                              ","            0.0","          100.0"
000025,"aiAustrittTemperatur                           ","AI: Austritt Temperatur                                    ","°C                             ","          -30.0","           70.0"
000026,"aiAustrittFeuchte                              ","AI: Austritt rel. Feuchte                                  ","%                              ","            0.0","          100.0"
000027,"aoDrehzahlvorgVentilator1                      ","AO: Drehzahlvorgabe Ventilator 1                           ","%                              ","            0.0","          100.0"
000028,"aoDrehzahlvorgVentilator2                      ","AO: Drehzahlvorgabe Ventilator 2                           ","%                              ","            0.0","          100.0"
000029,"aoDrehzahlvorgKompressorModul1                 ","AO: Drehzahlvorgabe Kompressor Modul 1                     ","%                              ","            0.0","          100.0"
000030,"aoDrehzahlvorgKompressorModul2                 ","AO: Drehzahlvorgabe Kompressor Modul 2                     ","%                              ","            0.0","          100.0"
000031,"aoLeistungsvorgHeizregister                    ","AO: Drehzahlvorgabe Heizregister                           ","%                              ","            0.0","          100.0"
000032,"aoTemperaturvorgWarmluftofen                   ","AO: Temperaturvorgabe Warmluftofen                         ","°C                             ","            0.0","          100.0"
000033,"aoDrehzahlvorgAbluftventilator                 ","AO: Drehzahlvorgabe Abluftventilator                       ","%                              ","            0.0","          100.0"
000034,"gMindestlaufzOelsumpfOk                        ","ALLG: Laufzeit Oelsumpfheizung OK                          ","0/1                            ","              0","              1"
000035,"gStatusAnlage.LuftmengeAktuell                 ","ALLG: Luftmenge Aktuell                                    ","m³/h                           ","            0.0","      9999999.9"
000036,"di24VDCinternIstOk                             ","Status DI Absicherung 24VDC                                ","0/1                            ","              0","              1"
000037,"diNiederdruckOkModul1                          ","Status DI Niederdruck OK Modul 1                           ","0/1                            ","              0","              1"
000038,"diHochdruckOkModul1                            ","Status DI Hochdruck OK Modul 1                             ","0/1                            ","              0","              1"
000039,"diNiederdruckOkModul2                          ","Status DI Niederdruck OK Modul 2                           ","0/1                            ","              0","              1"
000040,"diHochdruckOkModul2                            ","Status DI Hochdruck OK Modul 2                             ","0/1                            ","              0","              1"
000041,"diKopftempKompressorModul1                     ","Status DI Kopftemperatur Kompressor Modul 1                ","0/1                            ","              0","              1"
000042,"diKopftempKompressorModul2                     ","Status DI Kopftemperatur Kompressor Modul 2                ","0/1                            ","              0","              1"
000043,"diOeldruckKompressorModul1                     ","Status DI Öldruck Kompressor Modul 1                       ","0/1                            ","              0","              1"
000044,"diOeldruckKompressorModul2                     ","Status DI Öldruck Kompressor Modul 2                       ","0/1                            ","              0","              1"
000045,"diVollschutzKompressorModul1                   ","Status DI Vollschutz Kompressor Modul 1                    ","0/1                            ","              0","              1"
000046,"diVollschutzKompressorModul2                   ","Status DI Vollschutz Kompressor Modul 2                    ","0/1                            ","              0","              1"
000047,"diBetriebsmldgKompressorModul1                 ","Status DI Betriebsmeldung FU Kompressor Modul 1            ","0/1                            ","              0","              1"
000048,"diBetriebsmldgKompressorModul2                 ","Status DI Betriebsmeldung FU Kompressor Modul 2            ","0/1                            ","              0","              1"
000049,"diAnfEntfeuchterExtern                         ","Status DI Anforderung Entfeuchter Extern                   ","0/1                            ","              0","              1"
000050,"diLeistungsvorgKompressorExtMod1               ","Status DI Leistungsvorgabe Extern Modul 1                  ","0/1                            ","              0","              1"
000051,"diVentilator1InBetrieb                         ","Status DI Betriebsmeldung Ventilator 1                     ","0/1                            ","              0","              1"
000052,"diVentilator2InBetrieb                         ","Status DI Betriebsmeldung Ventilator 2                     ","0/1                            ","              0","              1"
000053,"diDrehzahlbegrVentilator1                      ","Status DI Drehzahlbegrenzung Ventilator 1                  ","0/1                            ","              0","              1"
000054,"diDrehzahlbegrVentilator2                      ","Status DI Drehzahlbegrenzung Ventilator 2                  ","0/1                            ","              0","              1"
000055,"diScheitholzofenInBetrieb                      ","Status DI Betriebsmeldung Scheitholzofen                   ","0/1                            ","              0","              1"
000056,"diWarmluftofenInBetrieb                        ","Status DI Betriebsmeldung Warmluftofen                     ","0/1                            ","              0","              1"
000057,"diNotstromaggregatInBetrieb                    ","Status DI Betriebsmeldung Notstromaggregat                 ","0/1                            ","              0","              1"
000058,"diBox1Offen                                    ","Status DI Klappe Box 1 Offen                               ","0/1                            ","              0","              1"
000059,"diBox1Geschl                                   ","Status DI Klappe Box 1 Geschlossen                         ","0/1                            ","              0","              1"
000060,"diBox2Offen                                    ","Status DI Klappe Box 2 Offen                               ","0/1                            ","              0","              1"
000061,"diBox2Geschl                                   ","Status DI Klappe Box 2 Geschlossen                         ","0/1                            ","              0","              1"
000062,"diBox3Offen                                    ","Status DI Klappe Box 3 Offen                               ","0/1                            ","              0","              1"
000063,"diBox3Geschl                                   ","Status DI Klappe Box 3 Geschlossen                         ","0/1                            ","              0","              1"
000064,"diBox4Offen                                    ","Status DI Klappe Box 4 Offen                               ","0/1                            ","              0","              1"
000065,"diBox4Geschl                                   ","Status DI Klappe Box 4 Geschlossen                         ","0/1                            ","              0","              1"
000066,"diBox5Offen                                    ","Status DI Klappe Box 5 Offen                               ","0/1                            ","              0","              1"
000067,"diBox5Geschl                                   ","Status DI Klappe Box 5 Geschlossen                         ","0/1                            ","              0","              1"
000068,"diBox6Offen                                    ","Status DI Klappe Box 6 Offen                               ","0/1                            ","              0","              1"
000069,"diBox6Geschl                                   ","Status DI Klappe Box 6 Geschlossen                         ","0/1                            ","              0","              1"
000070,"diBypassklappeOffen                            ","Status DI Bypassklappe Offen                               ","0/1                            ","              0","              1"
000071,"diBypassklappeGeschl                           ","Status DI Bypassklappe Geschlossen                         ","0/1                            ","              0","              1"
000072,"diUmschaltklappe1Offen                         ","Status DI Umschaltklappe 1 Offen                           ","0/1                            ","              0","              1"
000073,"diUmschaltklappe2Offen                         ","Status DI Umschaltklappe 2 Offen                           ","0/1                            ","              0","              1"
000074,"diUmschaltklappe1Geschl                        ","Status DI Umschaltklappe 1 Geschlossen                     ","0/1                            ","              0","              1"
000075,"diUmschaltklappe2Geschl                        ","Status DI Umschaltklappe 2 Geschlossen                     ","0/1                            ","              0","              1"
000076,"diAbluftklappeOffen                            ","Status DI Abluftklappe Offen                               ","0/1                            ","              0","              1"
000077,"diAbluftklappeGeschl                           ","Status DI Abluftklappe Geschlossen                         ","0/1                            ","              0","              1"
000078,"diAbluftventInBetrieb                          ","Status DI Abluftventilator in Betrieb                      ","0/1                            ","              0","              1"
000079,"doTrocknungInBetrieb                           ","Status DO Trocknung in Betrieb                             ","0/1                            ","              0","              1"
000080,"doTrocknungStoerung                            ","Status DO Trocknung Störung                                ","0/1                            ","              0","              1"
000081,"doWarmluftofenEin                              ","Status DO Freigabe Warmluftofen                            ","0/1                            ","              0","              1"
000082,"doHeizregisterEin                              ","Status DO Freigabe Heizregister                            ","0/1                            ","              0","              1"
000083,"doKompressorEinModul1                          ","Status DO Freigabe Kompressor Modul 1                      ","0/1                            ","              0","              1"
000084,"doKompressorEinModul2                          ","Status DO Freigabe Kompressor Modul 2                      ","0/1                            ","              0","              1"
000085,"doMagnetventilEinModul1                        ","Status DO Magnetventil Modul 1                             ","0/1                            ","              0","              1"
000086,"doMagnetventilEinModul2                        ","Status DO Freigabe Magnetventil Modul 2                    ","0/1                            ","              0","              1"
000087,"doOelsumpfheizungEinModul1                     ","Status DO Ölsumpfheizung Modul 1                           ","0/1                            ","              0","              1"
000088,"doOelsumpfheizungEinModul2                     ","Status DO Freigabe Ölsumpfheizung Modul 2                  ","0/1                            ","              0","              1"
000089,"doVentilator1Ein                               ","Status DO Freigabe Ventilator 1                            ","0/1                            ","              0","              1"
000090,"doVentilator2Ein                               ","Status DO Freigabe Ventilator 2                            ","0/1                            ","              0","              1"
000091,"doNotstromaggregatEin                          ","Status DO Freigabe Notstromaggregat                        ","0/1                            ","              0","              1"
000092,"doBypassklappeOeffnen                          ","Status DO Bypassklappe Freigabe                            ","0/1                            ","              0","              1"
000093,"doAbluftklappeFreigabe                         ","Status DO Abluftklappe Freigabe                            ","0/1                            ","              0","              1"
000094,"doAbluftventilatorEin                          ","Status DO Freigabe Abluftventilator                        ","0/1                            ","              0","              1"
000095,"doUmluftklappe1Freigabe                        ","Status DO Umluftklappe 1 Freigabe                          ","0/1                            ","              0","              1"
000096,"doUmluftklappe2Freigabe                        ","Status DO Umluftklappe 2 Freigabe                          ","0/1                            ","              0","              1"
000097,"doFreigabeBox1                                 ","Status DO Boxenklappe 1 Öffnen                             ","0/1                            ","              0","              1"
000098,"doFreigabeBox2                                 ","Status DO Boxenklappe 2 Öffnen                             ","0/1                            ","              0","              1"
000099,"doFreigabeBox3                                 ","Status DO Boxenklappe 3 Öffnen                             ","0/1                            ","              0","              1"
000100,"doFreigabeBox4                                 ","Status DO Boxenklappe 4 Öffnen                             ","0/1                            ","              0","              1"
000101,"doFreigabeBox5                                 ","Status DO Boxenklappe 5 Öffnen                             ","0/1                            ","              0","              1"
000102,"doFreigabeBox6                                 ","Status DO Boxenklappe 6 Öffnen                             ","0/1                            ","              0","              1"
000103,"doBrandschutzklappeAuf                         ","Status DO Brandschutzklappe Öffnen                         ","0/1                            ","              0","              1"
000104,"doAbluftklappeFreigabe                         ","Status DO Abluftklappe Öffnen                              ","0/1                            ","              0","              1"
000105,"doAbluftventilatorEin                          ","Status DO Abluftventilator Ein                             ","0/1                            ","              0","              1"
000106,"Nutzungsdaten.BstGes.Kompressor1Std            ","Betriebsstunden Gesamt: Kompressor 1                       ","h                              ","              0","        9999999"
000107,"Nutzungsdaten.BstGes.Kompressor2Std            ","Betriebsstunden Gesamt: Kompressor 2                       ","h                              ","              0","        9999999"
000108,"Nutzungsdaten.BstGes.Ventilator1Std            ","Betriebsstunden Gesamt: Ventilator 1                       ","h                              ","              0","        9999999"
000109,"Nutzungsdaten.BstGes.Ventilator2Std            ","Betriebsstunden Gesamt: Ventilator 2                       ","h                              ","              0","        9999999"
000110,"Nutzungsdaten.BstGes.WarmluftofenStd           ","Betriebsstunden Gesamt: Warmluftofen                       ","h                              ","              0","        9999999"
000111,"Nutzungsdaten.BstGes.HeizregisterStd           ","Betriebsstunden Gesamt: Heizregister                       ","h                              ","              0","        9999999"
000112,"Nutzungsdaten.BstGes.Box1Std                   ","Betriebsstunden Gesamt: Box 1                              ","h                              ","              0","        9999999"
000113,"Nutzungsdaten.BstGes.Box2Std                   ","Betriebsstunden Gesamt: Box 2                              ","h                              ","              0","        9999999"
000114,"Nutzungsdaten.BstGes.Box3Std                   ","Betriebsstunden Gesamt: Box 3                              ","h                              ","              0","        9999999"
000115,"Nutzungsdaten.BstGes.Box4Std                   ","Betriebsstunden Gesamt: Box 4                              ","h                              ","              0","        9999999"
000116,"Nutzungsdaten.BstGes.Box5Std                   ","Betriebsstunden Gesamt: Box 5                              ","h                              ","              0","        9999999"
000117,"Nutzungsdaten.BstGes.Box6Std                   ","Betriebsstunden Gesamt: Box 6                              ","h                              ","              0","        9999999"
000118,"Nutzungsdaten.BstGes.OelsumpfheizungStd        ","Betriebsstunden Gesamt: Oelsumpfheizung                    ","h                              ","              0","        9999999"
000119,"Nutzungsdaten.BstGes.Abtauung1Std              ","Betriebsstunden Gesamt: Abtauung Modul 1                   ","h                              ","              0","        9999999"
000120,"Nutzungsdaten.BstGes.Abtauung2Std              ","Betriebsstunden Gesamt: Abtauung Modul 2                   ","h                              ","              0","        9999999"
000121,"Nutzungsdaten.BstGes.AbluftventStd             ","Betriebsstunden Gesamt: Abluftventilator                   ","h                              ","              0","        9999999"
000122,"Nutzungsdaten.BstGes.FrischluftbetrStd         ","Betriebsstunden Gesamt: Frischluftbetrieb                  ","h                              ","              0","        9999999"
000123,"Nutzungsdaten.BstGes.UmluftbetrStd             ","Betriebsstunden Gesamt: Umluftbetrieb                      ","h                              ","              0","        9999999"
000124,"Nutzungsdaten.Energiemessung.LeistungAktuell   ","Energiemessung: Leistung Aktuell                           ","kW                             ","            0.0","        99999.9"
000125,"Nutzungsdaten.Energiemessung.EnergieTag        ","Energiemessung: Energie Tag                                ","kWh                            ","            0.0","      9999999.9"
000126,"Nutzungsdaten.Energiemessung.EnergieGesamt     ","Energiemessung: Energie Gesamt                             ","kWh                            ","            0.0","      9999999.9"
000127,"gStatusAnlage.WetterIstSchlecht                ","ALLG: Wetter ist schlecht                                  ","0/1                            ","              0","              1"
000128,"doEntfFremdFreigabe                            ","Status DO Freigabe Entfeuchter Fremdgerät                  ","0/1                            ","              0","              1"
000129,"diEntfeuchterFremdInBetrieb                    ","Status DI Betriebsmldg Entfeuchter Fremdgerät              ","0/1                            ","              0","              1"
000130,"diEntfeuchterFremdStoerung                     ","Status DI Störmeldung Entfeuchter Fremdgerät               ","0/1                            ","              0","              1"
```

### InputOutput.var
```iecst
(*Digitale Ausgänge (DO) ===================================================================================================================================================*)
VAR
	doVentilator1Ein : BOOL;
	doVentilator2Ein : BOOL;
	doTrocknungInBetrieb : BOOL;
	doFreigabeBox1 : BOOL;
	doFreigabeBox2 : BOOL;
	doTrocknungStoerung : BOOL;
	doWarmluftofenEin : BOOL;
	doHeizregisterEin : BOOL;
	doFreigabeBox3 : BOOL;
	doFreigabeBox4 : BOOL;
	doFreigabeBox5 : BOOL;
	doFreigabeBox6 : BOOL;
	doBrandschutzklappeAuf : BOOL;
	doAbluftventilatorEin : BOOL;
	doAbluftklappeFreigabe : BOOL;
	doAbluftklappeOeffnen : BOOL; (*Nur bei 3.04 in Verwendung*)
	doAbluftklappeSchliessen : BOOL; (*Nur bei 3.04 in Verwendung*)
	doUmluftklappe2Schliessen : BOOL; (*Nur bei 3.04 in Verwendung*)
	doUmluftklappe2Oeffnen : BOOL; (*Nur bei 3.04 in Verwendung*)
	doUmluftklappe1Schliessen : BOOL; (*Nur bei 3.04 in Verwendung*)
	doUmluftklappe1Oeffnen : BOOL; (*Nur bei 3.04 in Verwendung*)
	doUmluftklappe1Freigabe : BOOL;
	doUmluftklappe2Freigabe : BOOL;
	doNotstromaggregatEin : BOOL;
	doKompressorEinModul1 : BOOL;
	doKompressorEinModul2 : BOOL;
	doMagnetventilEinModul1 : BOOL;
	doMagnetventilEinModul2 : BOOL;
	doOelsumpfheizungEinModul1 : BOOL;
	doOelsumpfheizungEinModul2 : BOOL;
	doBypassklappeSchliessen : BOOL; (*Nur bei 3.04 in Verwendung*)
	doBypassklappeOeffnen : BOOL;
	doEntfFremdFreigabe : BOOL; (*Nur bei HB4000 in Verwendung*)
	doLuftentfeuchterStrombegrEin : BOOL; (*Nur bei HB4000 in Verwendung*)
END_VAR
(*Analoge Ausgänge (AO) =====================================================================================================================================================*)
VAR
	aoDrehzahlvorgVentilator1 : REAL;
	aoTemperaturvorgWarmluftofen : REAL;
	aoDrehzahlvorgVentilator2 : REAL;
	aoLeistungsvorgHeizregister : REAL;
	aoDrehzahlvorgAbluftventilator : REAL;
	aoDrehzahlvorgKompressorModul1 : REAL;
	aoDrehzahlvorgKompressorModul2 : REAL;
END_VAR
(*Analoge Eingänge (AI) =====================================================================================================================================================*)
VAR
	aiFrischluftTemperatur : REAL;
	aiFrischluftFeuchte : REAL;
	aiTrockenluftTemperatur : REAL;
	aiTrockenluftFeuchte : REAL;
	aiAbluftTemperatur : REAL;
	aiAbluftFeuchte : REAL;
	aiDachluftTemperatur : REAL;
	aiDachluftFeuchte : REAL;
	aiLuftgeschwindigkeit : REAL;
	aiDifferenzdruck : REAL;
	aiNiederdruckModul2 : REAL;
	aiNiederdruckModul1 : REAL;
	aiHochdruckModul2 : REAL;
	aiHochdruckModul1 : REAL;
	aiEintrittTemperatur : REAL;
	aiEintrittFeuchte : REAL;
	aiAustrittTemperatur : REAL;
	aiAustrittFeuchte : REAL;
END_VAR
(*Digitale Eingänge (DI) =====================================================================================================================================================*)
VAR
	di230VACIstOk : BOOL; (*Nur bei HB4000 in Verwendung*)
	diEntfeuchterFremdInBetrieb : BOOL; (*Nur bei HB4000 in Verwendung*)
	diEntfeuchterFremdStoerung : BOOL; (*Nur bei HB4000 in Verwendung*)
	diTasteTrocknungPausieren : BOOL; (*Nur bei HB4000 in Verwendung*)
	diDrehfeldIstKorrekt : BOOL; (*Nur bei 3.04 in Verwendung*)
	diVentilator1InBetrieb : BOOL;
	di24VDCinternIstOk : BOOL;
	diBox1Offen : BOOL;
	diBox1Geschl : BOOL;
	diBox2Offen : BOOL;
	diBox2Geschl : BOOL;
	diVentilator2InBetrieb : BOOL;
	diDrehzahlbegrVentilator1 : BOOL;
	diDrehzahlbegrVentilator2 : BOOL;
	diScheitholzofenInBetrieb : BOOL;
	diWarmluftofenInBetrieb : BOOL;
	diBox3Offen : BOOL;
	diBox3Geschl : BOOL;
	diBox4Offen : BOOL;
	diBox4Geschl : BOOL;
	diBox5Offen : BOOL;
	diBox5Geschl : BOOL;
	diBox6Offen : BOOL;
	diBox6Geschl : BOOL;
	diAbluftventInBetrieb : BOOL;
	diAbluftklappeOffen : BOOL;
	diAbluftklappeGeschl : BOOL;
	diUmschaltklappe1Offen : BOOL;
	diUmschaltklappe1Geschl : BOOL;
	diUmschaltklappe2Offen : BOOL;
	diUmschaltklappe2Geschl : BOOL;
	diNotstromaggregatInBetrieb : BOOL;
	diNiederdruckOkModul1 : BOOL;
	diNiederdruckOkModul2 : BOOL;
	diHochdruckOkModul1 : BOOL;
	diHochdruckOkModul2 : BOOL;
	diKopftempKompressorModul1 : BOOL;
	diKopftempKompressorModul2 : BOOL;
	diOeldruckKompressorModul1 : BOOL;
	diOeldruckKompressorModul2 : BOOL;
	diVollschutzKompressorModul1 : BOOL;
	diVollschutzKompressorModul2 : BOOL;
	diBetriebsmldgKompressorModul1 : BOOL;
	diBetriebsmldgKompressorModul2 : BOOL;
	diAnfEntfeuchterExtern : BOOL;
	diLeistungsvorgKompressorExtMod1 : BOOL;
	diBypassklappeGeschl : BOOL;
	diBypassklappeOffen : BOOL;
END_VAR
(*Statuseingänge (DI) =====================================================================================================================================================*)
VAR
	diStatusNiederdruckMinMod1 : BOOL;
	diStatusNiederdruckMaxMod1 : BOOL;
	diStatusHochdruckMinMod1 : BOOL;
	diStatusHochdruckMaxMod1 : BOOL;
	diStatusNiederdruckMinMod2 : BOOL;
	diStatusNiederdruckMaxMod2 : BOOL;
	diStatusHochdruckMinMod2 : BOOL;
	diStatusHochdruckMaxMod2 : BOOL;
	diStatusDifferenzdruckMax : BOOL;
	diStatusDifferenzdruckMin : BOOL;
	diStatusLuftgeschwDrahtbruch : BOOL;
	diStatusLuftgeschwMax : BOOL;
	diStatusLuftgeschwMin : BOOL;
	diStatusEintrittTempMin : BOOL;
	diStatusEintrittTempMax : BOOL;
	diStatusEintrittFeuchteMin : BOOL;
	diStatusEintrittFeuchteMax : BOOL;
	diStatusAustrittTempMin : BOOL;
	diStatusAustrittTempMax : BOOL;
	diStatusAustrittFeuchteMin : BOOL;
	diStatusAustrittFeuchteMax : BOOL;
	diStatusFrischluftFeuchteMax : BOOL;
	diStatusFrischluftFeuchteMin : BOOL;
	diStatusFrischluftTempMax : BOOL;
	diStatusFrischluftTempMin : BOOL;
	diStatusTrockenluftFeuchteMax : BOOL;
	diStatusTrockenluftFeuchteMin : BOOL;
	diStatusTrockenluftTempMax : BOOL;
	diStatusTrockenluftTempMin : BOOL;
	diStatusDachluftFeuchteMax : BOOL;
	diStatusDachluftFeuchteMin : BOOL;
	diStatusDachluftTempMax : BOOL;
	diStatusDachluftTempMin : BOOL;
	diStatusAbluftTempMax : BOOL;
	diStatusAbluftTempMin : BOOL;
	diStatusAbluftFeuchteMax : BOOL;
	diStatusAbluftFeuchteMin : BOOL;
END_VAR
```

### Program Logical/IO/aktorenMapping
